FUNCTION_BLOCK Test_NotificationCount EXTENDS tcl_SimpleUnitTestLibrary.T_UnitTestBase
VAR
    Source   : T_Notification;
    Handler  : T_NotificationHandler;
    IsRaised : BOOL;
	Count : DINT;
END_VAR

Handler.FB_init(
    bInitRetains := FALSE,  
    bInCopyCode  := FALSE);

Source.ClearNotificationHandlers().AddNotificationHandler(Handler);

Source.Raise();
Source.Raise();
Source.Raise();
IsRaised := Handler.IsRaised(UnhandledNotificationsCount => Count);

Assertion.AssertEquals_BOOL(
    Expected     := TRUE,
    Actual       := IsRaised,
    VariableName := 'IsRaised');

Assertion.AssertEquals_DINT(
    Expected     := 3,
    Actual       := Count,
    VariableName := 'Count');

IsRaised := Handler.IsRaised(UnhandledNotificationsCount => Count);

Assertion.AssertEquals_BOOL(
    Expected     := FALSE,
    Actual       := IsRaised,
    VariableName := 'IsRaised');

Assertion.AssertEquals_DINT(
    Expected     := 0,
    Actual       := Count,
    VariableName := 'Count');


TestFinished();

END_FUNCTION_BLOCK

(* stored: Version 1.1.0.1, ProductVersion 3.1.4024.9
   POU Test_NotificationCount: Id {5a998e2d-812e-4528-950c-0f147306f34d}, SpecialFunc None *)
